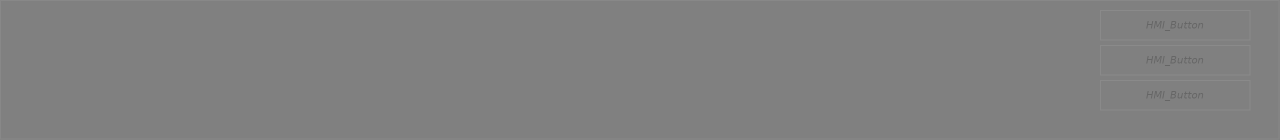
VISUALIZATION Header  // 1280x140
    Rectangle (0,0 1280x140)
    Frame (1100,10 150x30)
        shows HMI_Button(i_sText := 'Start', iq_stButton := GVL_Modules.g_fbHmiMachCtrlsManager.s_fbBtnReqStart.s_stHmi)
    Frame (1100,45 150x30)
        shows HMI_Button(i_sText := 'Stop', iq_stButton := GVL_Modules.g_fbHmiMachCtrlsManager.s_fbBtnReqStop.s_stHmi)
    Frame (1100,80 150x30)
        shows HMI_Button(i_sText := 'Reset', iq_stButton := GVL_Modules.g_fbHmiMachCtrlsManager.s_fbBtnReqReset.s_stHmi)
END_VISUALIZATION

(* stored: Version 1.1.0.1, ProductVersion 3.1.4026.13
   Visu Header: Id {a37fa97e-ff1b-4946-8bc8-0c4fc8751f6e} *)
